ABB RobotStudio station: Globe Picking & Placing.rspag

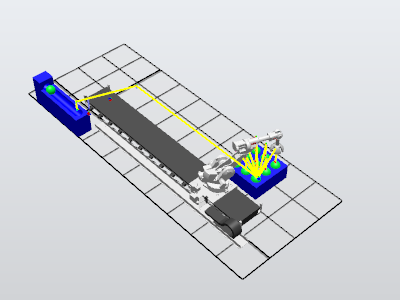
--- station ---
Station SimulationExam (saved by RobotStudio 24.3.10958.1)
Controller Controller1, task T_ROB1: task frame (RAPID world) sits at (395.5, 560, 374.5) mm in the station
Controller Controller1
  mechanical unit ROB_1: IRB4400_60_196__03, 6 joints, base frame (0, 0, 0) mm
  mechanical unit TRACK_1: IRBT4004_STD_0_0_6__04, 1 joints, base frame (0, 0, 0) mm
Layout (positions relative to the parent item):
  - IRB4400_60_196__03 [mechanism, from %ABB.RobotStudio.Models.IRB4400%\IRB4400_60_196_G_03.rslib] at (5395.5, 560, 374.5) mm; joint values [1.2088, 0.9435, 0.007, 0, 1.5638, -0.362] (rad or m)
  - IRBT4004_STD_0_0_6__04 [mechanism] at (0, 0, 0) mm; joint values [5] (rad or m)
      links: Base, Link1
  - globe_pallet [part] at (5000, 1200, 0) mm, size 1300 x 1300 x 500 mm
  - SC_globeTool [smart component] at (6033.51, 2244.83, 1580.77) mm, rotated rx 180 ry 0 rz -90 deg
      signals: DI diGrip, DO doGripped
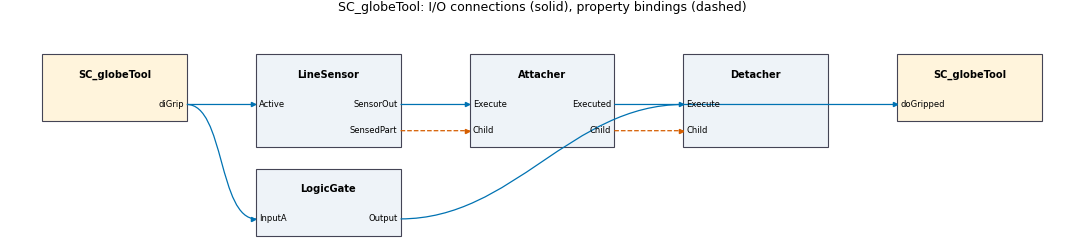
      connections:
        LineSensor.SensorOut -> Attacher.Execute
        SC_globeTool.diGrip -> LineSensor.Active
        SC_globeTool.diGrip -> LogicGate.InputA
        LogicGate.Output -> Detacher.Execute
        Attacher.Executed -> SC_globeTool.doGripped
        LineSensor.SensedPart => Attacher.Child
        Attacher.Child => Detacher.Child
    - globeTool [mechanism] at (0, 0, 0) mm
        TCP globeTool at (0, 0, 332.2) mm
        links: globe_tool
    - LogicGate [smart component, from Components\LogicGate.rslib]
        properties: Operator=NOT; Delay=0
    - Detacher [smart component, from Components\Detacher.rslib]
        properties: Child=globe_18; KeepPosition=true
    - Attacher [smart component, from Components\Attacher.rslib]
        properties: Parent=globeTool; Flange=0; Child=globe_18; Mount=false; Offset=[0 0 0]; Orientation=[0 0 0]
    - LineSensor [smart component, from Components\LineSensor.rslib]
        properties: Start=[0 0 0.35]; End=[0 0 0.4]; Length=0.05; Radius=0.00135135135135135; Tag=(none); SensedPart=globe_18; SensedPoint=[6.03351025390625 2.2448271484375 0.61921728515625]
      - _sensorPart_ [part], size 2.7 x 2.7 x 50 mm
  - globe [part], size 299 x 298 x 300 mm
  - SC_Conveyor [smart component]
      signals: DI diRollBall, DO doBallRolled
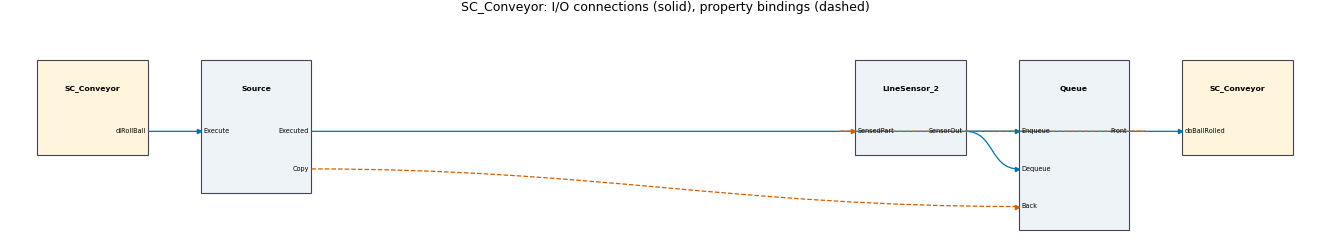
      connections:
        Source.Executed -> Queue.Enqueue
        LineSensor_2.SensorOut -> Queue.Dequeue
        SC_Conveyor.diRollBall -> Source.Execute
        LineSensor_2.SensorOut -> SC_Conveyor.doBallRolled
        Source.Copy => Queue.Back
        Queue.Front => LineSensor_2.SensedPart
    - globe_conveyour [part] at (-1500, -1000, 0) mm, rotated rx 90 ry 0 rz 90 deg, size 500 x 1000 x 2300 mm
    - LinearMover [smart component, from Components\LinearMover.rslib]
        properties: Object=Queue; Direction=[1 0 0]; Speed=0.5; Reference=Global; ReferenceObject=(none)
    - Source [smart component, from Components\Source.rslib]
        properties: Source=globe; Copy=globe_19; Parent=(none); Position=[0 0 0]; Orientation=[0 0 0]; Transient=false; PhysicsBehavior=0
    - Queue [smart component, from Components\Queue.rslib]
        properties: Back=globe_19; Front=globe_19; Queue={68c48d71-7424-40c7-bcb9-1e960fbf49b3};{792be63c-9d12-4e40-8aaf-e2b1b6aaaa99}; NumberOfObjects=1
    - LineSensor_2 [smart component, from Components\LineSensor.rslib]
        properties: Start=[0.7 -0.75 0.7]; End=[0.68 -0.75 0.7]; Length=0.02; Radius=0.00315315315315315; Tag=(none); SensedPart=(none); SensedPoint=[0 0 0]
      - _sensorPart_ [part], size 20 x 6.3 x 6.3 mm
  - globe_10 [part] at (4010.49, 689.4, -239) mm, rotated rx 0 ry 0 rz 180 deg, size 299 x 298 x 300 mm
  - globe_11 [part] at (4010.49, 1089.4, -229.87) mm, rotated rx 0 ry 0 rz -180 deg, size 299 x 298 x 300 mm
  - globe_12 [part] at (4010.49, 1489.4, -226.95) mm, rotated rx 0 ry 0 rz 180 deg, size 299 x 298 x 300 mm
  - globe_13 [part] at (4410.49, 1489.4, -236.31) mm, rotated rx 0 ry 0 rz 180 deg, size 299 x 298 x 300 mm
  - globe_14 [part] at (4410.49, 1089.4, -229.87) mm, rotated rx 0 ry 0 rz 180 deg, size 299 x 298 x 300 mm
  - globe_15 [part] at (4410.49, 689.4, -229.87) mm, rotated rx 0 ry 0 rz -180 deg, size 299 x 298 x 300 mm
  - globe_16 [part] at (4810.49, 689.4, -226.95) mm, rotated rx 0 ry 0 rz -180 deg, size 299 x 298 x 300 mm
  - globe_17 [part] at (4810.49, 1089.4, -229.87) mm, rotated rx 0 ry 0 rz 180 deg, size 299 x 298 x 300 mm
  - globe_18 [part] at (4810.49, 1489.4, -236.31) mm, rotated rx 0 ry 0 rz -180 deg, size 299 x 298 x 300 mm
  - globe_19 [part] at (324, 0, 0) mm, size 299 x 298 x 300 mm
Attachment: IRB4400_60_196__03 is attached to IRBT4004_STD_0_0_6__04 / Link1
Attachment: SC_globeTool is attached to IRB4400_60_196__03 / Link6
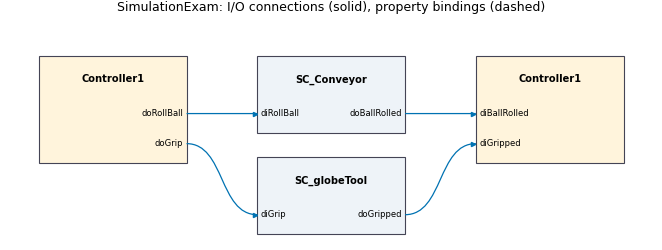
Station logic (signal -> signal, property => property):
  Controller1.doRollBall -> SC_Conveyor.diRollBall
  Controller1.doGrip -> SC_globeTool.diGrip
  SC_Conveyor.doBallRolled -> Controller1.diBallRolled
  SC_globeTool.doGripped -> Controller1.diGripped

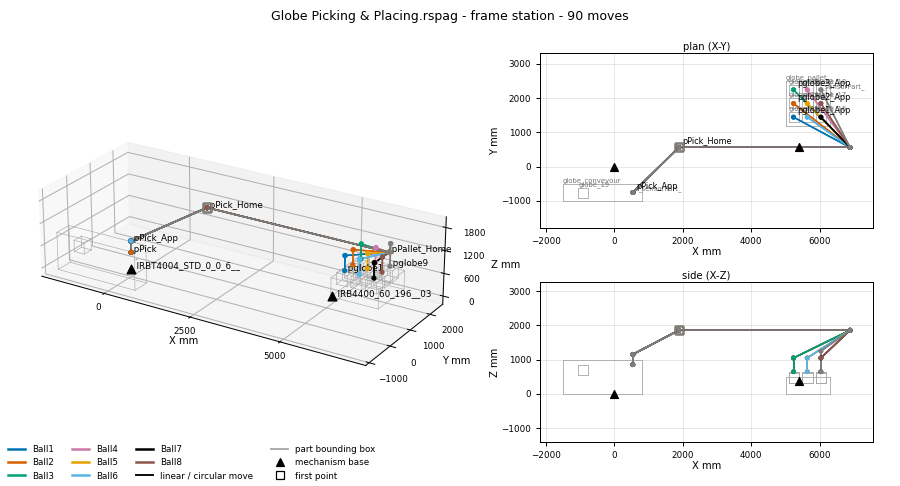
[picture p0: tool path of Globe Picking & Placing.rspag in frame station, 90 of 90 moves have a stored position in this frame; points joined in program order, loops and branches not executed]
--- Controller Data/Controller1/RAPID/TASK1/PROGMOD/CalibData.mod ---
MODULE CalibData
    PERS tooldata globeTool:=[TRUE,[[0,0,332.197],[1,0,0,0]],[1,[0,0,1],[1,0,0,0],0,0,0]];
ENDMODULE

--- Controller Data/Controller1/RAPID/TASK1/PROGMOD/MainModule.mod ---
MODULE MainModule
    TASK PERS wobjdata Workobject_conveyor:=[FALSE,TRUE,"",[[404.5,-1060,325.5],[0,-0.707106781,0.707106781,0]],[[0,0,0],[1,0,0,0]]];
    TASK PERS wobjdata Workobject_Pallet:=[FALSE,TRUE,"",[[4604.5,640,125.5],[0,0.707106781,0.707106781,0]],[[0,0,0],[1,0,0,0]]];
ENDMODULE

--- Controller Data/Controller1/RAPID/TASK1/PROGMOD/Module1.mod ---
MODULE Module1
        CONST robtarget pPick_Home:=[[-1060,-1084.434597591,-1158.4015],[0.612372436,0.353553391,-0.353553391,0.612372436],[-1,0,-1,0],[0,9E+09,9E+09,9E+09,9E+09,9E+09]];
    CONST robtarget pPick_App:=[[255.427,259.016,-453.658],[0,0,0,1],[-1,0,0,0],[0,9E+09,9E+09,9E+09,9E+09,9E+09]];
    CONST robtarget pPick:=[[255.427,259.016,-153.658],[0,0,0,1],[-1,0,0,0],[0,9E+09,9E+09,9E+09,9E+09,9E+09]];
    CONST robtarget pPallet_Home:=[[-640,1884.434597591,-1358.4015],[0.612372436,-0.353553391,-0.353553391,-0.612372436],[0,-1,0,0],[5000,9E+09,9E+09,9E+09,9E+09,9E+09]];
    CONST robtarget pglobe1_App:=[[244.827,233.51,-548.572],[0,0,0,1],[1,0,0,0],[5000,9E+09,9E+09,9E+09,9E+09,9E+09]];
    CONST robtarget pglobe1:=[[244.827,233.51,-148.572],[0,0,0,1],[1,0,0,0],[5000,9E+09,9E+09,9E+09,9E+09,9E+09]];
    CONST robtarget pglobe2_App:=[[644.827,233.51,-548.572],[0,0,0,1],[1,0,0,0],[5000,9E+09,9E+09,9E+09,9E+09,9E+09]];
    CONST robtarget pglobe2:=[[644.827,233.51,-148.572],[0,0,0,1],[1,0,0,0],[5000,9E+09,9E+09,9E+09,9E+09,9E+09]];
    CONST robtarget pglobe3_App:=[[1044.827,233.51,-548.572],[0,0,0,1],[1,0,0,0],[5000,9E+09,9E+09,9E+09,9E+09,9E+09]];
    CONST robtarget pglobe3:=[[1044.827,233.51,-148.572],[0,0,0,1],[1,0,0,0],[5000,9E+09,9E+09,9E+09,9E+09,9E+09]];
    CONST robtarget pglobe4_App:=[[1044.827,633.51,-548.572],[0,0,0,1],[0,0,-1,0],[5000,9E+09,9E+09,9E+09,9E+09,9E+09]];
    CONST robtarget pglobe4:=[[1044.827,633.51,-148.572],[0,0,0,1],[0,0,-1,0],[5000,9E+09,9E+09,9E+09,9E+09,9E+09]];
    CONST robtarget pglobe5_App:=[[644.827,633.51,-548.572],[0,0,0,1],[0,0,-1,0],[5000,9E+09,9E+09,9E+09,9E+09,9E+09]];
    CONST robtarget pglobe5:=[[644.827,633.51,-148.572],[0,0,0,1],[0,0,-1,0],[5000,9E+09,9E+09,9E+09,9E+09,9E+09]];
    CONST robtarget pglobe6_App:=[[244.827,633.51,-548.572],[0,0,0,1],[0,0,-1,0],[5000,9E+09,9E+09,9E+09,9E+09,9E+09]];
    CONST robtarget pglobe6:=[[244.827,633.51,-148.572],[0,0,0,1],[0,0,-1,0],[5000,9E+09,9E+09,9E+09,9E+09,9E+09]];
    CONST robtarget pglobe7_App:=[[244.827,1033.51,-548.572],[0,0,0,1],[0,0,-1,0],[5000,9E+09,9E+09,9E+09,9E+09,9E+09]];
    CONST robtarget pglobe7:=[[244.827,1033.51,-148.572],[0,0,0,1],[0,0,-1,0],[5000,9E+09,9E+09,9E+09,9E+09,9E+09]];
    CONST robtarget pglobe8_App:=[[644.827,1033.51,-548.572],[0,0,0,1],[0,0,-1,0],[5000,9E+09,9E+09,9E+09,9E+09,9E+09]];
    CONST robtarget pglobe8:=[[644.827,1033.51,-148.572],[0,0,0,1],[0,0,-1,0],[5000,9E+09,9E+09,9E+09,9E+09,9E+09]];
    CONST robtarget pglobe9_App:=[[1044.827,1033.51,-748.572],[0,0,0,1],[0,0,-1,0],[5000,9E+09,9E+09,9E+09,9E+09,9E+09]];
    CONST robtarget pglobe9:=[[1044.827,1033.51,-148.572],[0,0,0,1],[0,0,-1,0],[5000,9E+09,9E+09,9E+09,9E+09,9E+09]];
!***********************************************************
    !
    ! Module:  Module1
    !
    ! Description:
    !   <Insert description here>
    !
    ! Author: DELL
    !
    ! Version: 1.0
    !
    !***********************************************************


    !***********************************************************
    !
    ! Procedure main
    !
    !   This is the entry point of your program
    !
    !***********************************************************
    PROC main()
        VAR num i := 1;
        !Reset all doSiginals
        Reset doGrip;
        Reset doRollBall;

        ! Wait for DiStart to be 1
        WaitDI diStart, 1;

        ! Roll the Ball
        SetDO doRollBall, 1;
        WaitTime 3;

        WHILE i < 10 DO
            IF i = 1 THEN
                Reset doRollBall;
                Ball1;
                i := i + 1;
            ELSEIF i = 2 THEN
                Reset doRollBall;
                Ball2;
                i := i + 1;
            ELSEIF i = 3 THEN
                Reset doRollBall;
                Ball3;
                i := i + 1;
            ELSEIF i = 4 THEN
                Reset doRollBall;
                Ball4;
                i := i + 1;
            ELSEIF i = 5 THEN
                Reset doRollBall;
                Ball5;
                i := i + 1;
            ELSEIF i = 6 THEN
                Reset doRollBall;
                Ball6;
                i := i + 1;
            ELSEIF i = 7 THEN
                Reset doRollBall;
                Ball7;
                i := i + 1;
            ELSEIF i = 8 THEN
                Reset doRollBall;
                Ball8;
                i := i + 1;
            ELSEIF i = 9 THEN
                Reset doRollBall;
                Ball9;
                i := i + 1;
            ENDIF
        ENDWHILE
    ENDPROC
    PROC Ball1()
        MoveL pPick_Home,v1500,z0,globeTool\WObj:=Workobject_conveyor;
        MoveL pPick_App,v1500,z0,globeTool\WObj:=Workobject_conveyor;
        MoveL pPick,v800,fine,globeTool\WObj:=Workobject_conveyor;
        SetDO doGrip, 1;
        WaitTime 1;
        MoveL pPick_App,v800,fine,globeTool\WObj:=Workobject_conveyor;
        MoveL pPick_Home,v1500,z0,globeTool\WObj:=Workobject_conveyor;
        MoveL pPallet_Home,v1500,z0,globeTool\WObj:=Workobject_Pallet;
        MoveL pglobe1_App,v1500,z0,globeTool\WObj:=Workobject_Pallet;
        MoveL pglobe1,v800,fine,globeTool\WObj:=Workobject_Pallet;
        SetDO doGrip, 0;
        WaitTime 1;
        MoveL pglobe1_App,v1500,z0,globeTool\WObj:=Workobject_Pallet;
        MoveL pPallet_Home,v1500,z0,globeTool\WObj:=Workobject_Pallet;
        SetDO doRollBall, 1;
    ENDPROC
    PROC Ball2()
        MoveL pPick_Home,v1500,z0,globeTool\WObj:=Workobject_conveyor;
        MoveL pPick_App,v1500,z0,globeTool\WObj:=Workobject_conveyor;
        MoveL pPick,v800,fine,globeTool\WObj:=Workobject_conveyor;
        SetDO doGrip, 1;
        WaitTime 1;
        MoveL pPick_App,v1500,z0,globeTool\WObj:=Workobject_conveyor;
        MoveL pPick_Home,v1500,z0,globeTool\WObj:=Workobject_conveyor;
        MoveL pPallet_Home,v1500,z0,globeTool\WObj:=Workobject_Pallet;
        MoveL pglobe2_App,v1500,z0,globeTool\WObj:=Workobject_Pallet;
        MoveL pglobe2,v800,fine,globeTool\WObj:=Workobject_Pallet;
        SetDO doGrip, 0;
        WaitTime 1;
        MoveL pglobe2_App,v1500,z0,globeTool\WObj:=Workobject_Pallet;
        MoveL pPallet_Home,v1500,z0,globeTool\WObj:=Workobject_Pallet;
        SetDO doRollBall, 1;
    ENDPROC
    PROC Ball3()
        MoveL pPick_Home,v1500,z0,globeTool\WObj:=Workobject_conveyor;
        MoveL pPick_App,v1500,z0,globeTool\WObj:=Workobject_conveyor;
        MoveL pPick,v800,fine,globeTool\WObj:=Workobject_conveyor;
        SetDO doGrip, 1;
        WaitTime 1;
        MoveL pPick_App,v1500,z0,globeTool\WObj:=Workobject_conveyor;
        MoveL pPick_Home,v1500,z0,globeTool\WObj:=Workobject_conveyor;
        MoveL pPallet_Home,v1500,z0,globeTool\WObj:=Workobject_Pallet;
        MoveL pglobe3_App,v1500,z0,globeTool\WObj:=Workobject_Pallet;
        MoveL pglobe3,v800,fine,globeTool\WObj:=Workobject_Pallet;
        SetDO doGrip, 0;
        WaitTime 1;
        MoveL pglobe3_App,v1500,z0,globeTool\WObj:=Workobject_Pallet;
        MoveL pPallet_Home,v1500,z0,globeTool\WObj:=Workobject_Pallet;
        SetDO doRollBall, 1;
    ENDPROC
    PROC Ball4()
        MoveL pPick_Home,v1500,z0,globeTool\WObj:=Workobject_conveyor;
        MoveL pPick_App,v1500,z0,globeTool\WObj:=Workobject_conveyor;
        MoveL pPick,v800,fine,globeTool\WObj:=Workobject_conveyor;
        SetDO doGrip, 1;
        WaitTime 1;
        MoveL pPick_App,v1500,z0,globeTool\WObj:=Workobject_conveyor;
        MoveL pPick_Home,v1500,z0,globeTool\WObj:=Workobject_conveyor;
        MoveL pPallet_Home,v1500,z0,globeTool\WObj:=Workobject_Pallet;
        MoveL pglobe4_App,v1500,z0,globeTool\WObj:=Workobject_Pallet;
        MoveL pglobe4,v800,fine,globeTool\WObj:=Workobject_Pallet;
        SetDO doGrip, 0;
        WaitTime 1;
        MoveL pglobe4_App,v1500,z0,globeTool\WObj:=Workobject_Pallet;
        MoveL pPallet_Home,v1500,z0,globeTool\WObj:=Workobject_Pallet;
        SetDO doRollBall, 1;
    ENDPROC
    PROC Ball5()
        MoveL pPick_Home,v1500,z0,globeTool\WObj:=Workobject_conveyor;
        MoveL pPick_App,v1500,z0,globeTool\WObj:=Workobject_conveyor;
        MoveL pPick,v800,fine,globeTool\WObj:=Workobject_conveyor;
        SetDO doGrip, 1;
        WaitTime 1;
        MoveL pPick_App,v1500,z0,globeTool\WObj:=Workobject_conveyor;
        MoveL pPick_Home,v1500,z0,globeTool\WObj:=Workobject_conveyor;
        MoveL pPallet_Home,v1500,z0,globeTool\WObj:=Workobject_Pallet;
        MoveL pglobe5_App,v1500,z0,globeTool\WObj:=Workobject_Pallet;
        MoveL pglobe5,v800,fine,globeTool\WObj:=Workobject_Pallet;
        SetDO doGrip, 0;
        WaitTime 1;
        MoveL pglobe5_App,v1500,z0,globeTool\WObj:=Workobject_Pallet;
        MoveL pPallet_Home,v1500,z0,globeTool\WObj:=Workobject_Pallet;
        SetDO doRollBall, 1;
    ENDPROC
    PROC Ball6()
        MoveL pPick_Home,v1500,z0,globeTool\WObj:=Workobject_conveyor;
        MoveL pPick_App,v1500,z0,globeTool\WObj:=Workobject_conveyor;
        MoveL pPick,v800,fine,globeTool\WObj:=Workobject_conveyor;
        SetDO doGrip, 1;
        WaitTime 1;
        MoveL pPick_App,v1500,z0,globeTool\WObj:=Workobject_conveyor;
        MoveL pPick_Home,v1500,z0,globeTool\WObj:=Workobject_conveyor;
        MoveL pPallet_Home,v1500,z0,globeTool\WObj:=Workobject_Pallet;
        MoveL pglobe6_App,v1500,z0,globeTool\WObj:=Workobject_Pallet;
        MoveL pglobe6,v800,fine,globeTool\WObj:=Workobject_Pallet;
        SetDO doGrip, 0;
        WaitTime 1;
        MoveL pglobe6_App,v1500,z0,globeTool\WObj:=Workobject_Pallet;
        MoveL pPallet_Home,v1500,z0,globeTool\WObj:=Workobject_Pallet;
        SetDO doRollBall, 1;
    ENDPROC
    PROC Ball7()
        MoveL pPick_Home,v1500,z0,globeTool\WObj:=Workobject_conveyor;
        MoveL pPick_App,v1500,z0,globeTool\WObj:=Workobject_conveyor;
        MoveL pPick,v800,fine,globeTool\WObj:=Workobject_conveyor;
        SetDO doGrip, 1;
        WaitTime 1;
        MoveL pPick_App,v1500,z0,globeTool\WObj:=Workobject_conveyor;
        MoveL pPick_Home,v1500,z0,globeTool\WObj:=Workobject_conveyor;
        MoveL pPallet_Home,v1500,z0,globeTool\WObj:=Workobject_Pallet;
        MoveL pglobe7_App,v1500,z0,globeTool\WObj:=Workobject_Pallet;
        MoveL pglobe7,v800,fine,globeTool\WObj:=Workobject_Pallet;
        SetDO doGrip, 0;
        WaitTime 1;
        MoveL pglobe7_App,v1500,z0,globeTool\WObj:=Workobject_Pallet;
        MoveL pPallet_Home,v1500,z0,globeTool\WObj:=Workobject_Pallet;
        SetDO doRollBall, 1;
    ENDPROC
    PROC Ball8()
        MoveL pPick_Home,v1500,z0,globeTool\WObj:=Workobject_conveyor;
        MoveL pPick_App,v1500,z0,globeTool\WObj:=Workobject_conveyor;
        MoveL pPick,v800,fine,globeTool\WObj:=Workobject_conveyor;
        SetDO doGrip, 1;
        WaitTime 1;
        MoveL pPick_App,v1500,z0,globeTool\WObj:=Workobject_conveyor;
        MoveL pPick_Home,v1500,z0,globeTool\WObj:=Workobject_conveyor;
        MoveL pPallet_Home,v1500,z0,globeTool\WObj:=Workobject_Pallet;
        MoveL pglobe8_App,v1500,z0,globeTool\WObj:=Workobject_Pallet;
        MoveL pglobe8,v800,fine,globeTool\WObj:=Workobject_Pallet;
        SetDO doGrip, 0;
        WaitTime 1;
        MoveL pglobe8_App,v1500,z0,globeTool\WObj:=Workobject_Pallet;
        MoveL pPallet_Home,v1500,z0,globeTool\WObj:=Workobject_Pallet;
        SetDO doRollBall, 1;
    ENDPROC
    PROC Ball9()
        MoveL pPick_Home,v1500,z0,globeTool\WObj:=Workobject_conveyor;
        MoveL pPick_App,v1500,z0,globeTool\WObj:=Workobject_conveyor;
        MoveL pPick,v800,fine,globeTool\WObj:=Workobject_conveyor;
        SetDO doGrip, 1;
        WaitTime 1;
        MoveL pPick_App,v1500,z0,globeTool\WObj:=Workobject_conveyor;
        MoveL pPick_Home,v1500,z0,globeTool\WObj:=Workobject_conveyor;
        MoveL pPallet_Home,v1500,z0,globeTool\WObj:=Workobject_Pallet;
        MoveL pglobe9_App,v1500,z0,globeTool\WObj:=Workobject_Pallet;
        MoveL pglobe9,v800,fine,globeTool\WObj:=Workobject_Pallet;
        SetDO doGrip, 0;
        WaitTime 1;
        MoveL pglobe9_App,v1500,z0,globeTool\WObj:=Workobject_Pallet;
        MoveL pPallet_Home,v1500,z0,globeTool\WObj:=Workobject_Pallet;
        SetDO doRollBall, 1;
    ENDPROC
ENDMODULE

--- Controller Data/Controller1/SYSPAR/EIO.cfg ---
EIO:CFG_1.0:6:1::
#
INDUSTRIAL_NETWORK:

      -Name "PROFIBUS" -Label "PROFIBUS Controller Network"\
      -CfgPath "HOME/pbus_cfg.bin"
#
PROFIBUS_DEVICE:

      -Name "Board10"
#
EIO_SIGNAL:

      -Name "doRollBall" -SignalType "DO" -Device "Board10" -DeviceMap "0"

      -Name "diBallRolled" -SignalType "DI" -Device "Board10" -DeviceMap "1"

      -Name "diStart" -SignalType "DI" -Device "Board10" -DeviceMap "2"

      -Name "doGrip" -SignalType "DO" -Device "Board10" -DeviceMap "3"

      -Name "diGripped" -SignalType "DI" -Device "Board10" -DeviceMap "4"
